Staubli VAL3: Programmetest.pgx

program Programmetest()
begin
  wait(EntreePower==true)
  movej(jJointRx[0],tTool,mNomSpeed)
  movej(jJointRx[1],tTool,mNomSpeed)
  waitEndMove()
end
